FUNCTION_BLOCK FB_Chamber1Endpoint1DoorCloseService EXTENDS FB_ServiceBase
VAR_INPUT
	IsDoorClose : BOOL;
	IsRobotInChamber : BOOL;
END_VAR
VAR_IN_OUT
	DoorCloseCtrl : BOOL;
END_VAR

M_UpdateService(CompletionBehavior := E_ServiceCompletionBehavior.NaturalCompletion);

METHOD PROTECTED H_OnExecute : E_PackMLHookResult
VAR_INPUT
	bFirstScan : BOOL;
END_VAR
H_OnExecute := E_PackMLHookResult.Busy;

DoorCloseCtrl := TRUE;

IF IsDoorClose = TRUE THEN
	H_OnExecute := E_PackMLHookResult.Done;
END_IF
END_METHOD

METHOD PROTECTED H_OnStarting : RobustSolution_BATW.E_PackMLHookResult
VAR_INPUT
	bFirstScan	: BOOL;
END_VAR
IF IsRobotInChamber THEN
	M_AddError( MainErrorId:= E_Chamber1ErrorCode.Close_Door_While_Robot_In_Chamber, SourceErrorId:= 0, Message:= 'Close door while robot in chamber.');
	RequestCommand(E_PackMLCommand.Stop);
END_IF
END_METHOD

END_FUNCTION_BLOCK

(* stored: Version 1.1.0.1, ProductVersion 3.1.4026.18
   POU FB_Chamber1Endpoint1DoorCloseService: Id {d8f384c9-dbfe-48a0-a93a-0c4f93ef162b}, SpecialFunc None
   Folder StateAction: Id {d6718092-13db-412c-a9a2-e9ff38355be8}
   Method H_OnExecute: Id {932ce45f-f47d-46af-8179-4c8f87fe1fb0}
   Method H_OnStarting: Id {47b05317-2dea-4db5-b9a1-f89c1f4d0532} *)
